// TIA Portal V16 export
// export: Created 2022-07-21T09:35:34.9401302Z, ExportSetting WithDefaults, DisplayName Totally Integrated Automation Portal, DisplayVersion V16 Update 4, DisplayName TIA Portal Version Control Interface, DisplayVersion V16 Update 2, DisplayName TIA Portal Openness, DisplayVersion V16 Update 4, DisplayName SINAMICS Startdrive Advanced, DisplayVersion V16 Update 5, DisplayName SINAMICS Startdrive G130, G150, S120, S150, SINAMICS MV, S210, DisplayVersion V16 Update 5, DisplayName SINAMICS Startdrive G110M, G120, G120C, G120D, G120P, G115D, DisplayVersion V16 Update 5, DisplayName STEP 7 Professional, DisplayVersion V16 Update 4, DisplayName STEP 7 Safety, DisplayVersion V16, DisplayName WinCC Advanced, DisplayVersion V16 Update 4
FUNCTION_BLOCK "fbVacuum"   // FB7, LAD
TITLE = Ejector / Blok funkcyjny edżektora
{ S7_Optimized_Access := 'TRUE' }
AUTHOR : a32thzz
VERSION : 0.1
// stored: AutoNumber false, IsIECCheckEnabled false, IsRetainMemResEnabled false, MemoryReserve 100, SetENOAutomatically false, UDAEnableTagReadback false
   VAR_INPUT
      generalRelease : Bool;   // Zezwolenie na pracę od warunków sprzętowych / General release
      autoVacuum : Bool;   // Aktywacja zasysania w trybie automatycznym / Activate vacuum in automatic mode
      fbkSensor : Bool := true;
      keepPartParameter : Bool := true;
      delayPTAlm0 : Time := T#1s;   // Czas opóźnienia dla alarmu 0 / delay alarm 0
      delayPTAlm1 : Time := T#1s;   // Czas opóźnienia dla alarmu 1 / delay alarm 1
      delayPTAlm2 : Time := T#1s;   // Czas opóźnienia dla alarmu 2 / delay alarm 2
      delayPTAlm3 : Time := T#1s;   // Czas opóźnienia dla alarmu 3 / delay alarm 3
      delayPTAlm4 : Time := T#1s;   // Czas opóźnienia dla alarmu 4 / delay alarm 4
      delayPTAlm5 : Time := T#1s;   // Czas opóźnienia dla alarmu 5 / delay alarm 5
      delayPTAlm6 : Time := T#1s;   // Czas opóźnienia dla alarmu 6 / delay alarm 6
      delayPTAlm7 : Time := T#1s;   // Czas opóźnienia dla alarmu 7 / delay alarm 7
      group : "typeGroup";   // Grupa do której przypisany jest edżektor / Ejector group
   END_VAR
   VAR_OUTPUT
      vacVacuum : Bool;   // Elektrozawór dla pozycji roboczej / Electrovalve for work position
   END_VAR
   VAR_IN_OUT
      vacuumTube : "typeVacuum";
   END_VAR
   VAR
      instTmrDlyAlm0 { S7_SetPoint := 'True'} : TON_TIME;   // Opóźnienie dla alarmu 0 / delay alarm 0
      instTmrDlyAlm1 { S7_SetPoint := 'True'} : TON_TIME;   // Opóźnienie dla alarmu 1 / delay alarm 1
      instTmrDlyAlm2 { S7_SetPoint := 'True'} : TON_TIME;   // Opóźnienie dla alarmu 2 / delay alarm 2
      instTmrDlyAlm3 { S7_SetPoint := 'True'} : TON_TIME;   // Opóźnienie dla alarmu 3 / delay alarm 3
      instTmrDlyAlm4 { S7_SetPoint := 'True'} : TON_TIME;   // Opóźnienie dla alarmu 4 / delay alarm 4
      instTmrDlyAlm5 { S7_SetPoint := 'True'} : TON_TIME;   // Opóźnienie dla alarmu 5 / delay alarm 5
      instTmrDlyAlm6 { S7_SetPoint := 'True'} : TON_TIME;   // Opóźnienie dla alarmu 6 / delay alarm 6
      instTmrDlyAlm7 { S7_SetPoint := 'True'} : TON_TIME;   // Opóźnienie dla alarmu 7 / delay alarm 7
      autoVacuumCmdMem { S7_SetPoint := 'True'} : Bool;   // Zasysanie zażądane w trybie ręcznym - bit pamięci / Vacuum requested in manual mode - memory bit
      handVacuumCmdMem { S7_SetPoint := 'True'} : Bool;   // Zasysanie zażądane w trybie ręcznym - bit pamięci / Vacuum requested in manual mode - memory bit
   END_VAR
   // instTmrDlyAlm0.PT := T#0ms;
   // instTmrDlyAlm1.PT := T#0ms;
   // instTmrDlyAlm2.PT := T#0ms;
   // instTmrDlyAlm3.PT := T#0ms;
   // instTmrDlyAlm4.PT := T#0ms;
   // instTmrDlyAlm5.PT := T#0ms;
   // instTmrDlyAlm6.PT := T#0ms;
   // instTmrDlyAlm7.PT := T#0ms;
BEGIN

REGION Network 1: No active alarms / Brak aktywnych alarmów
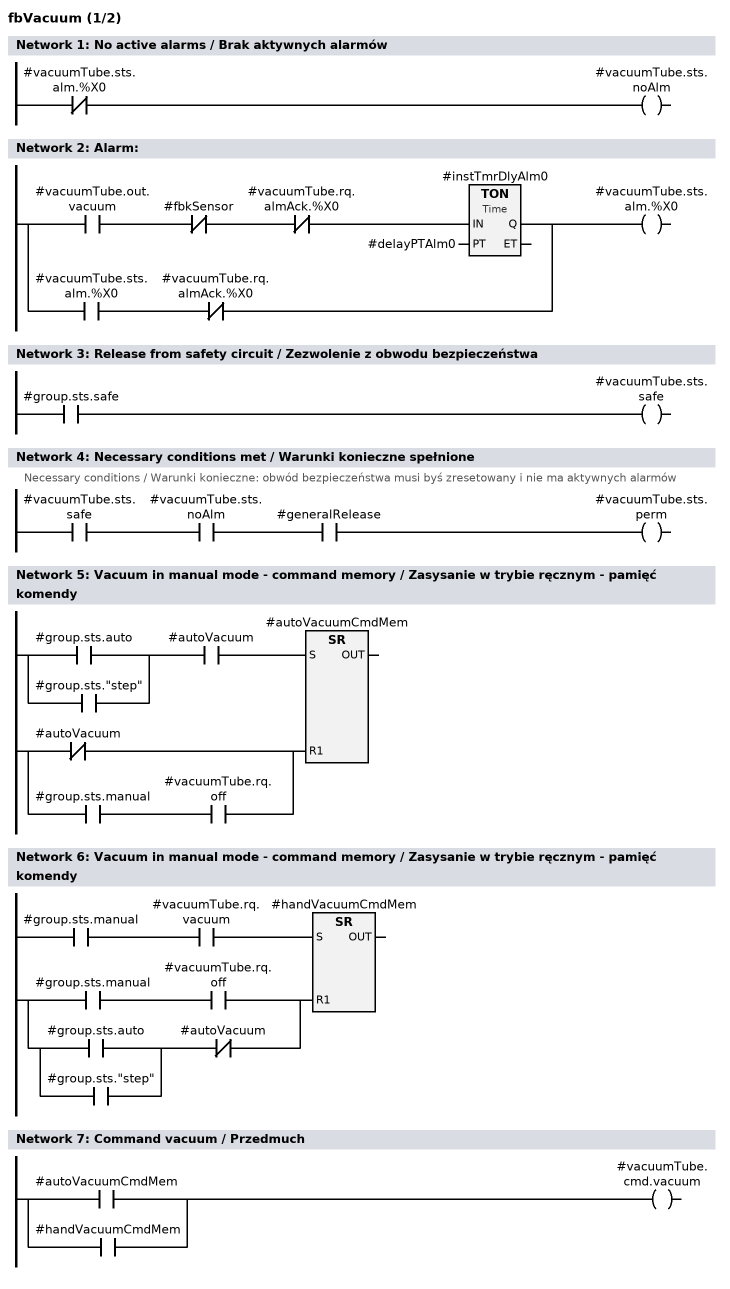
   RUNG wire#powerrail
      I_Contact( #vacuumTube.sts.alm.%X0 )
      Coil( #vacuumTube.sts.noAlm )
   END_RUNG
   // the same network as SCL:
   #vacuumTube.sts.noAlm := NOT #vacuumTube.sts.alm.%X0;
END_REGION

REGION Network 2: Alarm:
   RUNG wire#powerrail
      Contact( #vacuumTube.out.vacuum )
      I_Contact( #fbkSensor )
      I_Contact( #vacuumTube.rq.almAck.%X0 )
      { S7_Templates := "time_type := Time" } #instTmrDlyAlm0.TON(pt := #delayPTAlm0, et =>)
      wire#w1
      Coil( #vacuumTube.sts.alm.%X0 )
   END_RUNG
   RUNG wire#powerrail
      Contact( #vacuumTube.sts.alm.%X0 )
      I_Contact( #vacuumTube.rq.almAck.%X0 )
   END_RUNG wire#w1
   // the same network as SCL:
   #instTmrDlyAlm0(IN := #vacuumTube.out.vacuum AND NOT #fbkSensor AND NOT #vacuumTube.rq.almAck.%X0,   // TON
                   PT := #delayPTAlm0);
   #vacuumTube.sts.alm.%X0 := #instTmrDlyAlm0.Q OR (#vacuumTube.sts.alm.%X0 AND NOT #vacuumTube.rq.almAck.%X0);
END_REGION

REGION Network 3: Release from safety circuit / Zezwolenie z obwodu bezpieczeństwa
   RUNG wire#powerrail
      Contact( #group.sts.safe )
      Coil( #vacuumTube.sts.safe )
   END_RUNG
   // the same network as SCL:
   #vacuumTube.sts.safe := #group.sts.safe;
END_REGION

REGION Network 4: Necessary conditions met / Warunki konieczne spełnione
   // Necessary conditions / Warunki konieczne: obwód bezpieczeństwa musi byś zresetowany i nie ma aktywnych alarmów
   RUNG wire#powerrail
      Contact( #vacuumTube.sts.safe )
      Contact( #vacuumTube.sts.noAlm )
      Contact( #generalRelease )
      Coil( #vacuumTube.sts.perm )
   END_RUNG
   // the same network as SCL:
   #vacuumTube.sts.perm := #vacuumTube.sts.safe AND #vacuumTube.sts.noAlm AND #generalRelease;
END_REGION

REGION Network 5: Vacuum in manual mode - command memory / Zasysanie w trybie ręcznym - pamięć komendy
   RUNG wire#powerrail
      Contact( #group.sts.auto )
      wire#w1
      Contact( #autoVacuum )
      S_SR(operand := #autoVacuumCmdMem, r1 := wire#w2)
   END_RUNG
   RUNG wire#powerrail
      Contact( #group.sts."step" )
   END_RUNG wire#w1
   RUNG wire#powerrail
      I_Contact( #autoVacuum )
   END_RUNG wire#w2
   RUNG wire#powerrail
      Contact( #group.sts.manual )
      Contact( #vacuumTube.rq.off )
   END_RUNG wire#w2
   // the same network as SCL:
   IF (#group.sts.auto OR #group.sts."step") AND #autoVacuum THEN
       #autoVacuumCmdMem := TRUE;   // SR flip-flop
   END_IF;
   IF NOT #autoVacuum OR (#group.sts.manual AND #vacuumTube.rq.off) THEN #autoVacuumCmdMem := FALSE; END_IF;
END_REGION

REGION Network 6: Vacuum in manual mode - command memory / Zasysanie w trybie ręcznym - pamięć komendy
   RUNG wire#powerrail
      Contact( #group.sts.manual )
      Contact( #vacuumTube.rq.vacuum )
      S_SR(operand := #handVacuumCmdMem, r1 := wire#w2)
   END_RUNG
   RUNG wire#powerrail
      Contact( #group.sts.manual )
      Contact( #vacuumTube.rq.off )
   END_RUNG wire#w2
   RUNG wire#powerrail
      Contact( #group.sts.auto )
      wire#w1
      I_Contact( #autoVacuum )
   END_RUNG wire#w2
   RUNG wire#powerrail
      Contact( #group.sts."step" )
   END_RUNG wire#w1
   // the same network as SCL:
   IF #group.sts.manual AND #vacuumTube.rq.vacuum THEN
       #handVacuumCmdMem := TRUE;   // SR flip-flop
   END_IF;
   IF (#group.sts.manual AND #vacuumTube.rq.off) OR ((#group.sts.auto OR #group.sts."step") AND NOT #autoVacuum) THEN
       #handVacuumCmdMem := FALSE;
   END_IF;
END_REGION

REGION Network 7: Command vacuum / Przedmuch
   RUNG wire#powerrail
      Contact( #autoVacuumCmdMem )
      wire#w1
      Coil( #vacuumTube.cmd.vacuum )
   END_RUNG
   RUNG wire#powerrail
      Contact( #handVacuumCmdMem )
   END_RUNG wire#w1
   // the same network as SCL:
   #vacuumTube.cmd.vacuum := #autoVacuumCmdMem OR #handVacuumCmdMem;
END_REGION

REGION Network 8: Activate vacuum / Aktywacja zasysania
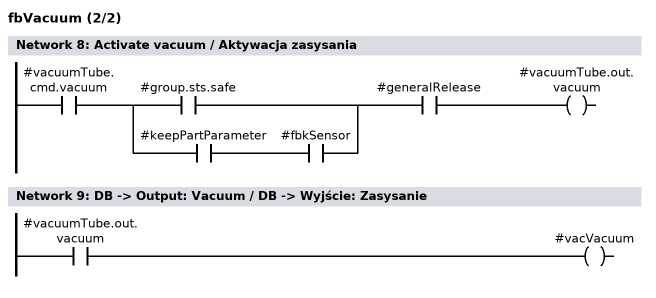
   RUNG wire#powerrail
      Contact( #vacuumTube.cmd.vacuum )
      wire#w1
      Contact( #group.sts.safe )
      wire#w2
      Contact( #generalRelease )
      Coil( #vacuumTube.out.vacuum )
   END_RUNG
   RUNG wire#w1
      Contact( #keepPartParameter )
      Contact( #fbkSensor )
   END_RUNG wire#w2
   // the same network as SCL:
   #vacuumTube.out.vacuum := #vacuumTube.cmd.vacuum AND (#group.sts.safe OR (#keepPartParameter AND #fbkSensor)) AND #generalRelease;
END_REGION

REGION Network 9: DB -> Output: Vacuum / DB -> Wyjście: Zasysanie
   RUNG wire#powerrail
      Contact( #vacuumTube.out.vacuum )
      Coil( #vacVacuum )
   END_RUNG
   // the same network as SCL:
   #vacVacuum := #vacuumTube.out.vacuum;
END_REGION
END_FUNCTION_BLOCK
